INTERFACE I_Enumerable EXTENDS T_QueryInterface

METHOD GetEnumerator : I_Enumerator
VAR_INPUT
END_VAR
END_METHOD

END_INTERFACE

(* stored: Version 1.1.0.1, ProductVersion 3.1.4024.4
   Itf I_Enumerable: Id {6eb14249-4d5f-4753-92bd-497beb404539}
   Method GetEnumerator: Id {b75ad828-4b10-4bd9-bf8f-17b35aa951aa} *)
